# EPICS substitutions: apps/CaenHVApp/Db/CaenHV_crate5.substitutions
# Third slot omited as no cables are connected to it
file "db/AS503_Chan.template" {
pattern
    {P,      H,  S,   V}
    {hchv,   5,  00,  000}
    {hchv,   5,  00,  001}
    {hchv,   5,  00,  002}
    {hchv,   5,  00,  003}
    {hchv,   5,  00,  004}
    {hchv,   5,  00,  005}
    {hchv,   5,  00,  006}
    {hchv,   5,  00,  007}
    {hchv,   5,  00,  008}
    {hchv,   5,  00,  009}
    {hchv,   5,  00,  010}
    {hchv,   5,  00,  011}
    {hchv,   5,  00,  012}
    {hchv,   5,  00,  013}
    {hchv,   5,  00,  014}
    {hchv,   5,  00,  015}
}
file "db/AS503_Chan.template" {
pattern
    {P,      H,  S,   V}
    {hchv,   5,  01, 000}
    {hchv,   5,  01, 001}
    {hchv,   5,  01, 002}
    {hchv,   5,  01, 003}
    {hchv,   5,  01, 004}
    {hchv,   5,  01, 005}
    {hchv,   5,  01, 006}
    {hchv,   5,  01, 007}
    {hchv,   5,  01, 008}
    {hchv,   5,  01, 009}
    {hchv,   5,  01, 010}
    {hchv,   5,  01, 011}
    {hchv,   5,  01, 012}
    {hchv,   5,  01, 013}
    {hchv,   5,  01, 014}
    {hchv,   5,  01, 015}
}
file "db/AS503_Chan.template" {
pattern
    {P,      H,  S,   V}
    {hchv,   5,  03, 000}
    {hchv,   5,  03, 001}
    {hchv,   5,  03, 002}
    {hchv,   5,  03, 003}
    {hchv,   5,  03, 004}
    {hchv,   5,  03, 005}
    {hchv,   5,  03, 006}
    {hchv,   5,  03, 007}
    {hchv,   5,  03, 008}
    {hchv,   5,  03, 009}
    {hchv,   5,  03, 010}
    {hchv,   5,  03, 011}
    {hchv,   5,  03, 012}
    {hchv,   5,  03, 013}
    {hchv,   5,  03, 014}
    {hchv,   5,  03, 015}
}
